// TIA Portal V19 export
FUNCTION_BLOCK "Common"   // FB13, FBD
TITLE = Common
{ S7_Optimized_Access := 'TRUE' }
AUTHOR : Siemens
// Common functions BeltLift
// stored: IsIECCheckEnabled true, MemoryReserve 100, SetENOAutomatically true
   VAR_INPUT
      autoStart { ExternalAccessible := 'False'; ExternalVisible := 'False'; ExternalWritable := 'False'} : Bool;
      autoStop { ExternalAccessible := 'False'; ExternalVisible := 'False'; ExternalWritable := 'False'} : Bool;
      plantOn { ExternalAccessible := 'False'; ExternalVisible := 'False'; ExternalWritable := 'False'} : Bool;
      seqStart { ExternalAccessible := 'False'; ExternalVisible := 'False'; ExternalWritable := 'False'} : Bool;
      posCaseBelt { ExternalAccessible := 'False'; ExternalVisible := 'False'; ExternalWritable := 'False'} : Int;
   END_VAR
   VAR_OUTPUT
      autoStarted { ExternalAccessible := 'False'; ExternalVisible := 'False'; ExternalWritable := 'False'} : Bool;
      autoStopped { ExternalAccessible := 'False'; ExternalVisible := 'False'; ExternalWritable := 'False'} : Bool;
   END_VAR
   VAR
      statCaseOnStopper { ExternalAccessible := 'False'; ExternalVisible := 'False'; ExternalWritable := 'False'} : Bool;
      statAutoStopped { ExternalAccessible := 'False'; ExternalVisible := 'False'; ExternalWritable := 'False'} : Bool;
   END_VAR
BEGIN

REGION Network 1
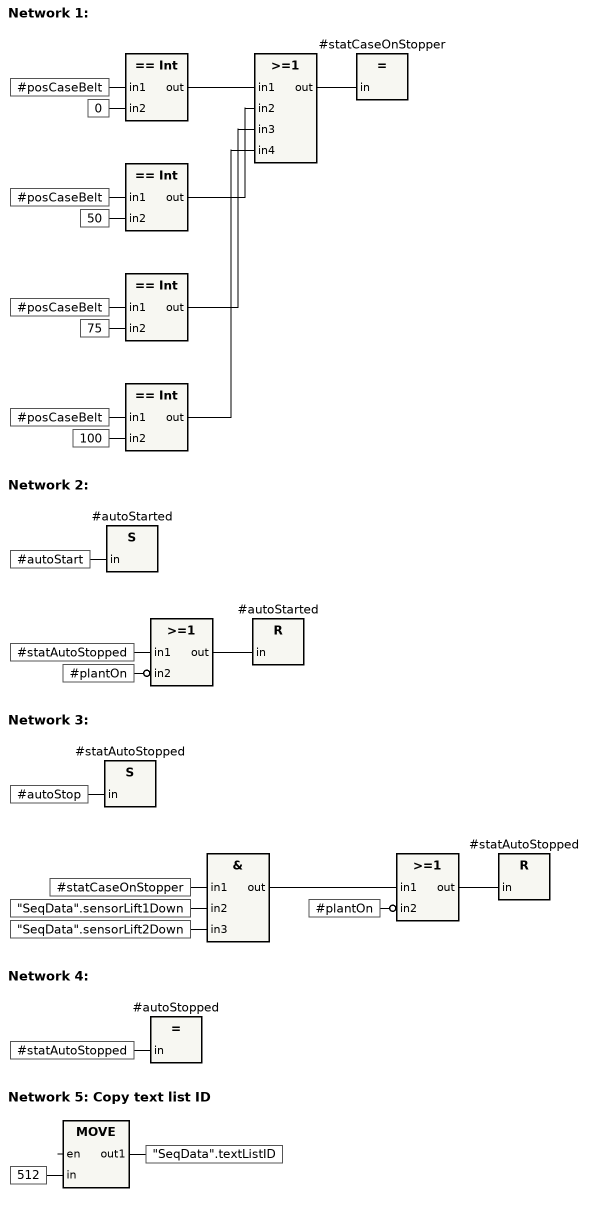
   #statCaseOnStopper := (#posCaseBelt = 0) OR (#posCaseBelt = 50) OR (#posCaseBelt = 75) OR (#posCaseBelt = 100);
END_REGION

REGION Network 2
   IF #autoStart THEN #autoStarted := TRUE; END_IF;
   IF #statAutoStopped OR NOT #plantOn THEN #autoStarted := FALSE; END_IF;
END_REGION

REGION Network 3
   IF #autoStop THEN #statAutoStopped := TRUE; END_IF;
   IF (#statCaseOnStopper AND "SeqData".sensorLift1Down AND "SeqData".sensorLift2Down) OR NOT #plantOn THEN
       #statAutoStopped := FALSE;
   END_IF;
END_REGION

REGION Network 4
   #autoStopped := #statAutoStopped;
END_REGION

REGION Network 5: Copy text list ID
   "SeqData".textListID := 512;
END_REGION
END_FUNCTION_BLOCK
